// TwinCAT 3 PLC project MAS418
// ProgramVersion: 3.1.4023.0
// libraries:
//   Tc2_Standard, * (Beckhoff Automation GmbH)
//   Tc2_System, * (Beckhoff Automation GmbH)
//   Tc3_Module, * (Beckhoff Automation GmbH)
// project tree:
//   DUTs/ E_Sensor.TcDUT
//   GVLs/ G_Task1.TcGVL
//   / PlcTask.TcTTO
//   POUs/ MAIN.TcPOU
// real-time tasks:
//   TASK PlcTask: cycle T#10ms, priority 20, ADS port 350
//   TASK PlcTask1: cycle T#10ms, priority 21, ADS port 351

CONFIGURATION MAS418
    RESOURCE PLC ON TwinCAT3
        TASK PlcTask(INTERVAL := T#10ms, PRIORITY := 21);
        PROGRAM MAIN WITH PlcTask : MAIN;
    END_RESOURCE
END_CONFIGURATION

// ---- DUTs/E_Sensor.TcDUT
{attribute 'qualified_only'}
{attribute 'strict'}
TYPE E_Sensor :
(
	Sick := 0,
	Pilz := 1,
	Parker := 2,
	Bosch := 3
);
END_TYPE

// ---- GVLs/G_Task1.TcGVL
{attribute 'qualified_only'}
VAR_GLOBAL
	tdTimeNowVar : TIME_OF_DAY := TOD#13:53:00.00;
	dDateVar : DATE := D#2023-02-07;
	tFiveSec : TIME := T#0D0H0M5S0MS;
	aArray : ARRAY[0..3] OF DATE := [D#2023-02-07, D#2023-02-08, D#2023-02-09, D#2023-02-10];
	etest : E_Sensor;
	bStartTimer: BOOL := FALSE;
	bOutput : BOOL := FALSE;
	fbTon : TON := ();
END_VAR

// ---- POUs/MAIN.TcPOU
PROGRAM MAIN
VAR
	pTimePointer : POINTER TO TIME_OF_DAY := ADR(G_Task1.tdTimeNowVar);
	pDatePointer : POINTER TO DATE := ADR(G_Task1.dDateVar);
	nReference : REFERENCE TO TIME REF= G_Task1.tFiveSec;
END_VAR

pTimePointer^ := TOD#18:37:12.47;
pDatePointer^ := D#2023-02-16;

nReference := T#0D0H0M1S0MS;

G_Task1.aArray[2] := D#2023-02-13;

G_Task1.etest := E_Sensor.Bosch;
G_Task1.bStartTimer := TRUE;
G_Task1.fbTon(IN:=G_Task1.bStartTimer, PT := T#10S);

END_PROGRAM
